Fanuc KAREL source: CLEAR.kl

PROGRAM T
%NOLOCKGROUP
VAR
 v0 : STRING[40]
 v1 : INTEGER
BEGIN
 CLEAR(v0, v1)
END T
